{attribute 'pack_mode' := '1'}
    {attribute 'OPC.UA.DA' := '1'}
    {attribute 'OPC.UA.DA.StructuredType' := '1'}
    (*
    ST_RW_BoolMb_HMI_IgnitionExp
    ==================================================
    Generated from Ignition UDT: RW_Bool_MB
    Total tags: 1
    Generated on: 2025-09-15 12:56:43
    *)
    TYPE ST_RW_BoolMb_HMI_IgnitionExp :
    STRUCT
        {attribute 'OPC.UA.DA' := '1'}
        {attribute 'OPC.UA.DA.Description' := '{Description}'}
        // {Description}
        Value : BOOL := FALSE;
    END_STRUCT
    END_TYPE

(* stored: Version 1.1.0.1
   DUT ST_RW_BoolMb_HMI_IgnitionExp: Id {1bb5bf68-3b78-4504-8101-fa80e5203203} *)
